{attribute 'qualified_only'}
VAR_GLOBAL
END_VAR

(* stored: Version 1.1.0.1, ProductVersion 3.1.4024.13
   GVL OpcuaData: Id {f250bad8-d97c-43c5-933e-b82ee7d7b261} *)
